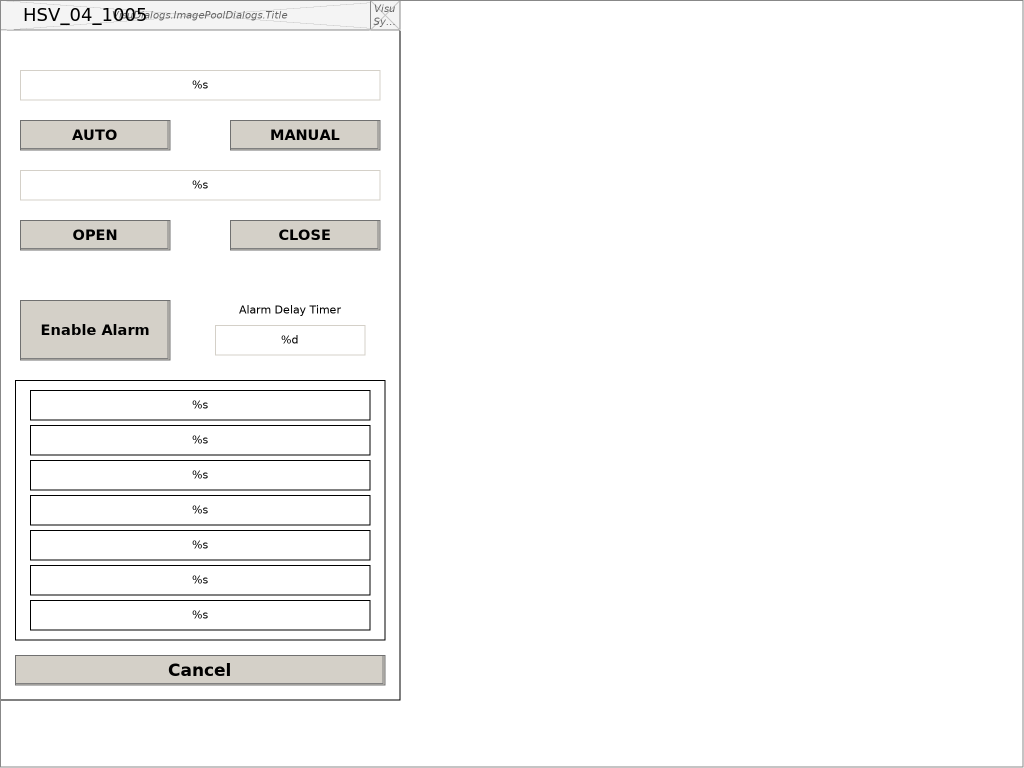
VISUALIZATION HSV_04_1005  // 1024x768
    Rectangle (0,0 400x700)
    Button (20,120 150x30), "AUTO"
        tap progHSVCntrl.HSV_04_1005.AutoReq
    Button (230,120 150x30), "MANUAL"
        tap progHSVCntrl.HSV_04_1005.ManReq
    Button (20,220 150x30), "OPEN"
        tap progHSVCntrl.HSV_04_1005.ManOpenReq
    Button (230,220 150x30), "CLOSE"
        tap progHSVCntrl.HSV_04_1005.ManCloseReq
    Textfield (20,70 360x30), "%s", text variable: progHSVCntrl.HSV_04_1005.strAutoMan
    Textfield (20,170 360x30), "%s", text variable: progHSVCntrl.HSV_04_1005.strOpenTravClose
    Button (20,300 150x60), "Enable Alarm"
        toggle progHSVCntrl.HSV_04_1005.EnableAlarm
    Textfield (215,325 150x30), "%d", text variable: progHSVCntrl.HSV_04_1005.AlarmDelayTime
    Label (215,295 150x30), "Alarm Delay Timer"
    Image (0,0 400x30), image: VisuDialogs.ImagePoolDialogs.Title
    Group (370,0 30x30)
        OnMouseClick: CloseDialog Dialog=HSV_04_1005, Result=OK, NumpadKeypadSet=True
        RoundedRectangle (0,0 30x30)
        Image (0,0 30x30), image: VisuSymbols.Symbols.Wrong
    Rectangle (15,380 370x260)
    RoundedRectangle (30,390 340x30), "%s", text variable: progHSVCntrl.HSV_04_1005.strInterlock_1
    RoundedRectangle (30,425 340x30), "%s", text variable: progHSVCntrl.HSV_04_1005.strInterlock_2
    RoundedRectangle (30,460 340x30), "%s", text variable: progHSVCntrl.HSV_04_1005.strInterlock_3
    RoundedRectangle (30,495 340x30), "%s", text variable: progHSVCntrl.HSV_04_1005.strInterlock_4
    RoundedRectangle (30,530 340x30), "%s", text variable: progHSVCntrl.HSV_04_1005.strInterlock_5
    RoundedRectangle (30,565 340x30), "%s", text variable: progHSVCntrl.HSV_04_1005.strInterlock_6
    RoundedRectangle (30,600 340x30), "%s", text variable: progHSVCntrl.HSV_04_1005.strInterlock_7
    Button (15,655 370x30), "Cancel"
        OnMouseClick: CloseDialog Dialog=HSV_04_1005, Result=OK, NumpadKeypadSet=True
    Label (20,0 210x30), "HSV_04_1005"
END_VISUALIZATION

(* stored: Version 1.1.0.1, ProductVersion 3.1.4022.17
   Visu HSV_04_1005: Id {3556cf42-4bb5-46d0-b7ed-6593ec304ad9} *)
